// TIA Portal V15.1 export
// export: Created 2024-05-17T05:38:27.533519Z, ExportSetting WithDefaults, DisplayName Totally Integrated Automation Portal, DisplayVersion V15.1 Update 5, DisplayName TIA Portal Openness, DisplayVersion V15.1 Update 5, DisplayName SINAMICS Startdrive Advanced, DisplayVersion V15.1, DisplayName G130, G150, S120, S150, SINAMICS MV, S210, DisplayVersion V15.1, DisplayName G110M, G120, G120C, G120D, G120P, DisplayVersion V15.1, DisplayName STEP 7 Professional, DisplayVersion V15.1 Update 5, DisplayName STEP 7 Safety, DisplayVersion V15.1, DisplayName WinCC Professional, DisplayVersion V15.1 Update 5, DisplayName SIMATIC Visualization Architect, DisplayVersion V15.1
FUNCTION "LETAFuseModule01_08_CPC20PN-Config" : Void   // FC1406, SCL
{ S7_Optimized_Access := 'TRUE' }
VERSION : 0.1
// stored: AutoNumber false, IsIECCheckEnabled false, SetENOAutomatically False, UDAEnableTagReadback false
   VAR_INPUT
      I_FuseMod1_Used : Bool;   // Fuse module is used
      I_FuseMod1_CH1_NominalCurrent : Int;   // Nominal current for the fuse
      I_FuseMod1_CH1_Name : String;   // Fuse name
      I_FuseMod1_CH1_Description : String;   // Description
      I_FuseMod1_CH2_NominalCurrent : Int;   // Nominal current for the fuse
      I_FuseMod1_CH2_Name : String;   // Fuse name
      I_FuseMod1_CH2_Description : String;   // Description
      I_FuseMod2_Used : Bool;   // Fuse module is used
      I_FuseMod2_CH1_NominalCurrent : Int;   // Nominal current for the fuse
      I_FuseMod2_CH1_Name : String;   // Fuse name
      I_FuseMod2_CH1_Description : String;   // Description
      I_FuseMod2_CH2_NominalCurrent : Int;   // Nominal current for the fuse
      I_FuseMod2_CH2_Name : String;   // Fuse name
      I_FuseMod2_CH2_Description : String;   // Description
      I_FuseMod3_Used : Bool;   // Fuse module is used
      I_FuseMod3_CH1_NominalCurrent : Int;   // Nominal current for the fuse
      I_FuseMod3_CH1_Name : String;   // Fuse name
      I_FuseMod3_CH1_Description : String;   // Description
      I_FuseMod3_CH2_NominalCurrent : Int;   // Nominal current for the fuse
      I_FuseMod3_CH2_Name : String;   // Fuse name
      I_FuseMod3_CH2_Description : String;   // Description
      I_FuseMod4_Used : Bool;   // Fuse module is used
      I_FuseMod4_CH1_NominalCurrent : Int;   // Nominal current for the fuse
      I_FuseMod4_CH1_Name : String;   // Fuse name
      I_FuseMod4_CH1_Description : String;   // Description
      I_FuseMod4_CH2_NominalCurrent : Int;   // Nominal current for the fuse
      I_FuseMod4_CH2_Name : String;   // Fuse name
      I_FuseMod4_CH2_Description : String;   // Description
      I_FuseMod5_Used : Bool;   // Fuse module is used
      I_FuseMod5_CH1_NominalCurrent : Int;   // Nominal current for the fuse
      I_FuseMod5_CH1_Name : String;   // Fuse name
      I_FuseMod5_CH1_Description : String;   // Description
      I_FuseMod5_CH2_NominalCurrent : Int;   // Nominal current for the fuse
      I_FuseMod5_CH2_Name : String;   // Fuse name
      I_FuseMod5_CH2_Description : String;   // Description
      I_FuseMod6_Used : Bool;   // Fuse module is used
      I_FuseMod6_CH1_NominalCurrent : Int;   // Nominal current for the fuse
      I_FuseMod6_CH1_Name : String;   // Fuse name
      I_FuseMod6_CH1_Description : String;   // Description
      I_FuseMod6_CH2_NominalCurrent : Int;   // Nominal current for the fuse
      I_FuseMod6_CH2_Name : String;   // Fuse name
      I_FuseMod6_CH2_Description : String;   // Description
      I_FuseMod7_Used : Bool;   // Fuse module is used
      I_FuseMod7_CH1_NominalCurrent : Int;   // Nominal current for the fuse
      I_FuseMod7_CH1_Name : String;   // Fuse name
      I_FuseMod7_CH1_Description : String;   // Description
      I_FuseMod7_CH2_NominalCurrent : Int;   // Nominal current for the fuse
      I_FuseMod7_CH2_Name : String;   // Fuse name
      I_FuseMod7_CH2_Description : String;   // Description
      I_FuseMod8_Used : Bool;   // Fuse module is used
      I_FuseMod8_CH1_NominalCurrent : Int;   // Nominal current for the fuse
      I_FuseMod8_CH1_Name : String;   // Fuse name
      I_FuseMod8_CH1_Description : String;   // Description
      I_FuseMod8_CH2_NominalCurrent : Int;   // Nominal current for the fuse
      I_FuseMod8_CH2_Name : String;   // Fuse name
      I_FuseMod8_CH2_Description : String;   // Description
   END_VAR
   VAR_IN_OUT
      IO_Config : "ETAFuseCPC20PNConfig";
   END_VAR
BEGIN
   #IO_Config.Fuse[1].Used := #I_FuseMod1_Used;
   #IO_Config.Fuse[1].NominalCurrent := #I_FuseMod1_CH1_NominalCurrent;
   #IO_Config.Fuse[1].Name := #I_FuseMod1_CH1_Name;
   #IO_Config.Fuse[1].Description := #I_FuseMod1_CH1_Description;

   #IO_Config.Fuse[2].Used := #I_FuseMod1_Used;
   #IO_Config.Fuse[2].NominalCurrent := #I_FuseMod1_CH2_NominalCurrent;
   #IO_Config.Fuse[2].Name := #I_FuseMod1_CH2_Name;
   #IO_Config.Fuse[2].Description := #I_FuseMod1_CH2_Description;

   #IO_Config.Fuse[3].Used := #I_FuseMod2_Used;
   #IO_Config.Fuse[3].NominalCurrent := #I_FuseMod2_CH1_NominalCurrent;
   #IO_Config.Fuse[3].Name := #I_FuseMod2_CH1_Name;
   #IO_Config.Fuse[3].Description := #I_FuseMod2_CH1_Description;

   #IO_Config.Fuse[4].Used := #I_FuseMod2_Used;
   #IO_Config.Fuse[4].NominalCurrent := #I_FuseMod2_CH2_NominalCurrent;
   #IO_Config.Fuse[4].Name := #I_FuseMod2_CH2_Name;
   #IO_Config.Fuse[4].Description := #I_FuseMod2_CH2_Description;

   #IO_Config.Fuse[5].Used := #I_FuseMod3_Used;
   #IO_Config.Fuse[5].NominalCurrent := #I_FuseMod3_CH1_NominalCurrent;
   #IO_Config.Fuse[5].Name := #I_FuseMod3_CH1_Name;
   #IO_Config.Fuse[5].Description := #I_FuseMod3_CH1_Description;

   #IO_Config.Fuse[6].Used := #I_FuseMod3_Used;
   #IO_Config.Fuse[6].NominalCurrent := #I_FuseMod3_CH2_NominalCurrent;
   #IO_Config.Fuse[6].Name := #I_FuseMod3_CH2_Name;
   #IO_Config.Fuse[6].Description := #I_FuseMod3_CH2_Description;

   #IO_Config.Fuse[7].Used := #I_FuseMod4_Used;
   #IO_Config.Fuse[7].NominalCurrent := #I_FuseMod4_CH1_NominalCurrent;
   #IO_Config.Fuse[7].Name := #I_FuseMod4_CH1_Name;
   #IO_Config.Fuse[7].Description := #I_FuseMod4_CH1_Description;

   #IO_Config.Fuse[8].Used := #I_FuseMod4_Used;
   #IO_Config.Fuse[8].NominalCurrent := #I_FuseMod4_CH2_NominalCurrent;
   #IO_Config.Fuse[8].Name := #I_FuseMod4_CH2_Name;
   #IO_Config.Fuse[8].Description := #I_FuseMod4_CH2_Description;

   #IO_Config.Fuse[9].Used := #I_FuseMod5_Used;
   #IO_Config.Fuse[9].NominalCurrent := #I_FuseMod5_CH1_NominalCurrent;
   #IO_Config.Fuse[9].Name := #I_FuseMod5_CH1_Name;
   #IO_Config.Fuse[9].Description := #I_FuseMod5_CH1_Description;

   #IO_Config.Fuse[10].Used := #I_FuseMod5_Used;
   #IO_Config.Fuse[10].NominalCurrent := #I_FuseMod5_CH2_NominalCurrent;
   #IO_Config.Fuse[10].Name := #I_FuseMod5_CH2_Name;
   #IO_Config.Fuse[10].Description := #I_FuseMod5_CH2_Description;

   #IO_Config.Fuse[11].Used := #I_FuseMod6_Used;
   #IO_Config.Fuse[11].NominalCurrent := #I_FuseMod6_CH1_NominalCurrent;
   #IO_Config.Fuse[11].Name := #I_FuseMod6_CH1_Name;
   #IO_Config.Fuse[11].Description := #I_FuseMod6_CH1_Description;

   #IO_Config.Fuse[12].Used := #I_FuseMod6_Used;
   #IO_Config.Fuse[12].NominalCurrent := #I_FuseMod6_CH2_NominalCurrent;
   #IO_Config.Fuse[12].Name := #I_FuseMod6_CH2_Name;
   #IO_Config.Fuse[12].Description := #I_FuseMod6_CH2_Description;

   #IO_Config.Fuse[13].Used := #I_FuseMod7_Used;
   #IO_Config.Fuse[13].NominalCurrent := #I_FuseMod7_CH1_NominalCurrent;
   #IO_Config.Fuse[13].Name := #I_FuseMod7_CH1_Name;
   #IO_Config.Fuse[13].Description := #I_FuseMod7_CH1_Description;

   #IO_Config.Fuse[14].Used := #I_FuseMod7_Used;
   #IO_Config.Fuse[14].NominalCurrent := #I_FuseMod7_CH2_NominalCurrent;
   #IO_Config.Fuse[14].Name := #I_FuseMod7_CH2_Name;
   #IO_Config.Fuse[14].Description := #I_FuseMod7_CH2_Description;

   #IO_Config.Fuse[15].Used := #I_FuseMod8_Used;
   #IO_Config.Fuse[15].NominalCurrent := #I_FuseMod8_CH1_NominalCurrent;
   #IO_Config.Fuse[15].Name := #I_FuseMod8_CH1_Name;
   #IO_Config.Fuse[15].Description := #I_FuseMod8_CH1_Description;

   #IO_Config.Fuse[16].Used := #I_FuseMod8_Used;
   #IO_Config.Fuse[16].NominalCurrent := #I_FuseMod8_CH2_NominalCurrent;
   #IO_Config.Fuse[16].Name := #I_FuseMod8_CH2_Name;
   #IO_Config.Fuse[16].Description := #I_FuseMod8_CH2_Description;
END_FUNCTION
